// Block: AreaXX_MatCounter_PERS

DATA_BLOCK AreaXX_MatCounter_PERS
VERSION : 0.1
   NON_RETAIN
   VAR
      PersistentValues : MatCountPersistent;
   END_VAR

BEGIN
   // No initialization required
END_DATA_BLOCK
